		(* CASE AT GLUE GOES FALSE WHEN AXIS IS MOVING AND MODULO GOES OUT OF RANGE *)
		IF (os_case_at_glue_latch OR ls_case_at_glue_latch)
			AND axis_is_moving(csp_case_transport_os_trailing.axis) 
			AND axis_get_actual_modulo_position(csp_case_transport_os_trailing.axis) > glue_trailing_upper_off //unlatch case at glue when past trailing glue flap window
			OR NOT axis_is_cam_engaged(csp_case_transport_os_trailing.axis)
			OR (csp.o_machine_is_stopped
			AND NOT axis_is_moving(csp_case_virtualMaster.axis))//unlatch on stop since glue will dry before closing
		THEN
			os_case_at_glue_latch := FALSE;
			ls_case_at_glue_latch := FALSE;
		END_IF
		
		IF toggle_shift_reg 
			AND	
			shift_register_step_has_status_item(
			step_id := case_at_glue_sr,
			status_bits_to_be_true := ITEM_HAS_LOAD,
			status_bits_to_be_false := 0,
			CONVERSION_this :=csp_case_main_statistics.sr)
		THEN 
			glue_shift_active :=TRUE;
		ELSE
			glue_shift_active :=FALSE;
		END_IF				
	
		
	(* RUN CONDITIONS *)
		IF run_conditions
			AND axis_is_moving(csp_case_transport_os_trailing.axis)
		THEN
			(* CHECKS PHASE WINDOWS TO DETERMINE IF GLUE GUN SHOULD BE ON *)
			
			(* OS UPPER DOTS *)
			IF os_case_at_glue_latch
				AND (
						(dot_1_enable AND phase_window_position_is_in_window(axis_get_actual_modulo_position(csp_case_transport_os_trailing.axis), os_leading_upper_dot_1_phwin)) (* LEADING UPPER DOT 1 *)
						OR (dot_2_enable AND phase_window_position_is_in_window(axis_get_actual_modulo_position(csp_case_transport_os_trailing.axis), os_leading_upper_dot_2_phwin)) (* LEADING UPPER DOT 2 *)
						OR (dot_3_enable AND phase_window_position_is_in_window(axis_get_actual_modulo_position(csp_case_transport_os_trailing.axis), os_leading_upper_dot_3_phwin)) (* LEADING UPPER DOT 3 *)
						OR (dot_4_enable AND phase_window_position_is_in_window(axis_get_actual_modulo_position(csp_case_transport_os_trailing.axis), os_leading_upper_dot_4_phwin)) (* LEADING UPPER DOT 4 *)
						OR (dot_5_enable AND phase_window_position_is_in_window(axis_get_actual_modulo_position(csp_case_transport_os_trailing.axis), os_leading_upper_dot_5_phwin)) (* LEADING UPPER DOT 5 *)
						OR (dot_6_enable AND phase_window_position_is_in_window(axis_get_actual_modulo_position(csp_case_transport_os_trailing.axis), os_leading_upper_dot_6_phwin)) (* LEADING UPPER DOT 6 *)
						OR (dot_1_enable AND phase_window_position_is_in_window(axis_get_actual_modulo_position(csp_case_transport_os_trailing.axis), os_trailing_upper_dot_1_phwin)) (* TRAILING UPPER DOT 1 *)
						OR (dot_2_enable AND phase_window_position_is_in_window(axis_get_actual_modulo_position(csp_case_transport_os_trailing.axis), os_trailing_upper_dot_2_phwin)) (* TRAILING UPPER DOT 2 *)
						OR (dot_3_enable AND phase_window_position_is_in_window(axis_get_actual_modulo_position(csp_case_transport_os_trailing.axis), os_trailing_upper_dot_3_phwin)) (* TRAILING UPPER DOT 3 *)
						OR (dot_4_enable AND phase_window_position_is_in_window(axis_get_actual_modulo_position(csp_case_transport_os_trailing.axis), os_trailing_upper_dot_4_phwin)) (* TRAILING UPPER DOT 4 *)
						OR (dot_5_enable AND phase_window_position_is_in_window(axis_get_actual_modulo_position(csp_case_transport_os_trailing.axis), os_trailing_upper_dot_5_phwin)) (* TRAILING UPPER DOT 5 *)
						OR (dot_6_enable AND phase_window_position_is_in_window(axis_get_actual_modulo_position(csp_case_transport_os_trailing.axis), os_trailing_upper_dot_6_phwin)) (* TRAILING UPPER DOT 6 *)
				)
				AND NOT os_upper_bypass_req
			THEN
					(* OS UPPER GUN 1 IF ENABLED *)
					IF os_upper_gun_1_enable
					THEN
						digital_output_set(os_upper_gun_1_do);
					END_IF
					(* OS UPPER GUN 2 IF ENABLED *)
					IF os_upper_gun_2_enable
					THEN
						digital_output_set(os_upper_gun_2_do);
					END_IF
			ELSE
				digital_output_reset(os_upper_gun_1_do);
				digital_output_reset(os_upper_gun_2_do);
			END_IF
			
			(* OS LOWER DOTS *)
			IF os_case_at_glue_latch
				AND (
						(dot_1_enable AND phase_window_position_is_in_window(axis_get_actual_modulo_position(csp_case_transport_os_trailing.axis), os_leading_lower_dot_1_phwin)) (* LEADING lower DOT 1 *)
						OR (dot_2_enable AND phase_window_position_is_in_window(axis_get_actual_modulo_position(csp_case_transport_os_trailing.axis), os_leading_lower_dot_2_phwin)) (* LEADING lower DOT 2 *)
						OR (dot_3_enable AND phase_window_position_is_in_window(axis_get_actual_modulo_position(csp_case_transport_os_trailing.axis), os_leading_lower_dot_3_phwin)) (* LEADING lower DOT 3 *)
						OR (dot_4_enable AND phase_window_position_is_in_window(axis_get_actual_modulo_position(csp_case_transport_os_trailing.axis), os_leading_lower_dot_4_phwin)) (* LEADING lower DOT 4 *)
						OR (dot_5_enable AND phase_window_position_is_in_window(axis_get_actual_modulo_position(csp_case_transport_os_trailing.axis), os_leading_lower_dot_5_phwin)) (* LEADING lower DOT 5 *)
						OR (dot_6_enable AND phase_window_position_is_in_window(axis_get_actual_modulo_position(csp_case_transport_os_trailing.axis), os_leading_lower_dot_6_phwin)) (* LEADING lower DOT 6 *)
						OR (dot_1_enable AND phase_window_position_is_in_window(axis_get_actual_modulo_position(csp_case_transport_os_trailing.axis), os_trailing_lower_dot_1_phwin)) (* TRAILING lower DOT 1 *)
						OR (dot_2_enable AND phase_window_position_is_in_window(axis_get_actual_modulo_position(csp_case_transport_os_trailing.axis), os_trailing_lower_dot_2_phwin)) (* TRAILING lower DOT 2 *)
						OR (dot_3_enable AND phase_window_position_is_in_window(axis_get_actual_modulo_position(csp_case_transport_os_trailing.axis), os_trailing_lower_dot_3_phwin)) (* TRAILING lower DOT 3 *)
						OR (dot_4_enable AND phase_window_position_is_in_window(axis_get_actual_modulo_position(csp_case_transport_os_trailing.axis), os_trailing_lower_dot_4_phwin)) (* TRAILING lower DOT 4 *)
						OR (dot_5_enable AND phase_window_position_is_in_window(axis_get_actual_modulo_position(csp_case_transport_os_trailing.axis), os_trailing_lower_dot_5_phwin)) (* TRAILING lower DOT 5 *)
						OR (dot_6_enable AND phase_window_position_is_in_window(axis_get_actual_modulo_position(csp_case_transport_os_trailing.axis), os_trailing_lower_dot_6_phwin)) (* TRAILING lower DOT 6 *)
				)
				AND NOT os_lower_bypass_req
			THEN
				(* OS LOWER GUN 1 IF ENABLED *)
				IF os_lower_gun_1_enable
				THEN
					digital_output_set(os_lower_gun_1_do);
				END_IF
				(* OS LOWER GUN 2 IF ENABLED *)
				IF os_lower_gun_2_enable
				THEN
					digital_output_set(os_lower_gun_2_do);
				END_IF
			ELSE
				digital_output_reset(os_lower_gun_1_do);
				digital_output_reset(os_lower_gun_2_do);
			END_IF
			
			
			(* LS UPPER DOTS *)
			IF ls_case_at_glue_latch
				AND (
						(dot_1_enable AND phase_window_position_is_in_window(axis_get_actual_modulo_position(csp_case_transport_ls_trailing.axis), ls_leading_upper_dot_1_phwin)) (* LEADING UPPER DOT 1 *)
						OR (dot_2_enable AND phase_window_position_is_in_window(axis_get_actual_modulo_position(csp_case_transport_ls_trailing.axis), ls_leading_upper_dot_2_phwin)) (* LEADING UPPER DOT 2 *)
						OR (dot_3_enable AND phase_window_position_is_in_window(axis_get_actual_modulo_position(csp_case_transport_ls_trailing.axis), ls_leading_upper_dot_3_phwin)) (* LEADING UPPER DOT 3 *)
						OR (dot_4_enable AND phase_window_position_is_in_window(axis_get_actual_modulo_position(csp_case_transport_ls_trailing.axis), ls_leading_upper_dot_4_phwin)) (* LEADING UPPER DOT 4 *)
						OR (dot_5_enable AND phase_window_position_is_in_window(axis_get_actual_modulo_position(csp_case_transport_ls_trailing.axis), ls_leading_upper_dot_5_phwin)) (* LEADING UPPER DOT 5 *)
						OR (dot_6_enable AND phase_window_position_is_in_window(axis_get_actual_modulo_position(csp_case_transport_ls_trailing.axis), ls_leading_upper_dot_6_phwin)) (* LEADING UPPER DOT 6 *)
						OR (dot_1_enable AND phase_window_position_is_in_window(axis_get_actual_modulo_position(csp_case_transport_ls_trailing.axis), ls_trailing_upper_dot_1_phwin)) (* TRAILING UPPER DOT 1 *)
						OR (dot_2_enable AND phase_window_position_is_in_window(axis_get_actual_modulo_position(csp_case_transport_ls_trailing.axis), ls_trailing_upper_dot_2_phwin)) (* TRAILING UPPER DOT 2 *)
						OR (dot_3_enable AND phase_window_position_is_in_window(axis_get_actual_modulo_position(csp_case_transport_ls_trailing.axis), ls_trailing_upper_dot_3_phwin)) (* TRAILING UPPER DOT 3 *)
						OR (dot_4_enable AND phase_window_position_is_in_window(axis_get_actual_modulo_position(csp_case_transport_ls_trailing.axis), ls_trailing_upper_dot_4_phwin)) (* TRAILING UPPER DOT 4 *)
						OR (dot_5_enable AND phase_window_position_is_in_window(axis_get_actual_modulo_position(csp_case_transport_ls_trailing.axis), ls_trailing_upper_dot_5_phwin)) (* TRAILING UPPER DOT 3 *)
						OR (dot_6_enable AND phase_window_position_is_in_window(axis_get_actual_modulo_position(csp_case_transport_ls_trailing.axis), ls_trailing_upper_dot_6_phwin)) (* TRAILING UPPER DOT 4 *)
				)
				AND NOT ls_upper_bypass_req
			THEN
				(* LS UPPER GUN 1 IF ENABLED *)
				IF ls_upper_gun_1_enable
				THEN
					digital_output_set(ls_upper_gun_1_do);
				END_IF
				(* LS UPPER GUN 2 IF ENABLED *)
				IF ls_upper_gun_2_enable
				THEN
					digital_output_set(ls_upper_gun_2_do);
				END_IF
			ELSE
				digital_output_reset(ls_upper_gun_1_do);
				digital_output_reset(ls_upper_gun_2_do);
			END_IF
			
			(* LS LOWER DOTS *)
			IF ls_case_at_glue_latch
				AND (
						(dot_1_enable AND phase_window_position_is_in_window(axis_get_actual_modulo_position(csp_case_transport_ls_trailing.axis), ls_leading_lower_dot_1_phwin)) (* LEADING lower DOT 1 *)
						OR (dot_2_enable AND phase_window_position_is_in_window(axis_get_actual_modulo_position(csp_case_transport_ls_trailing.axis), ls_leading_lower_dot_2_phwin)) (* LEADING lower DOT 2 *)
						OR (dot_3_enable AND phase_window_position_is_in_window(axis_get_actual_modulo_position(csp_case_transport_ls_trailing.axis), ls_leading_lower_dot_3_phwin)) (* LEADING lower DOT 3 *)
						OR (dot_4_enable AND phase_window_position_is_in_window(axis_get_actual_modulo_position(csp_case_transport_ls_trailing.axis), ls_leading_lower_dot_4_phwin)) (* LEADING lower DOT 4 *)
						OR (dot_5_enable AND phase_window_position_is_in_window(axis_get_actual_modulo_position(csp_case_transport_ls_trailing.axis), ls_leading_lower_dot_5_phwin)) (* LEADING lower DOT 5 *)
						OR (dot_6_enable AND phase_window_position_is_in_window(axis_get_actual_modulo_position(csp_case_transport_ls_trailing.axis), ls_leading_lower_dot_6_phwin)) (* LEADING lower DOT 6 *)
						OR (dot_1_enable AND phase_window_position_is_in_window(axis_get_actual_modulo_position(csp_case_transport_ls_trailing.axis), ls_trailing_lower_dot_1_phwin)) (* TRAILING lower DOT 1 *)
						OR (dot_2_enable AND phase_window_position_is_in_window(axis_get_actual_modulo_position(csp_case_transport_ls_trailing.axis), ls_trailing_lower_dot_2_phwin)) (* TRAILING lower DOT 2 *)
						OR (dot_3_enable AND phase_window_position_is_in_window(axis_get_actual_modulo_position(csp_case_transport_ls_trailing.axis), ls_trailing_lower_dot_3_phwin)) (* TRAILING lower DOT 3 *)
						OR (dot_4_enable AND phase_window_position_is_in_window(axis_get_actual_modulo_position(csp_case_transport_ls_trailing.axis), ls_trailing_lower_dot_4_phwin)) (* TRAILING lower DOT 4 *)
						OR (dot_5_enable AND phase_window_position_is_in_window(axis_get_actual_modulo_position(csp_case_transport_ls_trailing.axis), ls_trailing_lower_dot_5_phwin)) (* TRAILING lower DOT 3 *)
						OR (dot_6_enable AND phase_window_position_is_in_window(axis_get_actual_modulo_position(csp_case_transport_ls_trailing.axis), ls_trailing_lower_dot_6_phwin)) (* TRAILING lower DOT 4 *)
				)
				AND NOT ls_lower_bypass_req
			THEN
				(* LS LOWER GUN 1 IF ENABLED *)
				IF ls_lower_gun_1_enable
				THEN
					digital_output_set(ls_lower_gun_1_do);
				END_IF
				(* LS LOWER GUN 2 IF ENABLED *)
				IF ls_lower_gun_2_enable
				THEN
					digital_output_set(ls_lower_gun_2_do);
				END_IF
			ELSE
				digital_output_reset(ls_lower_gun_1_do);
				digital_output_reset(ls_lower_gun_2_do);
			END_IF
			
			
		ELSE (* LOST RUN CONDITIONS OR GLUE LATCH OR AXIS IS NOT MOVING *)
			(* OS GUNS RESET *)
			digital_output_reset(os_upper_gun_1_do);
			digital_output_reset(os_upper_gun_2_do);
			digital_output_reset(os_lower_gun_1_do);
			digital_output_reset(os_lower_gun_2_do);
			
			(* LS GUNS RESET *)
			digital_output_reset(ls_upper_gun_1_do);
			digital_output_reset(ls_upper_gun_2_do);
			digital_output_reset(ls_lower_gun_1_do);
			digital_output_reset(ls_lower_gun_2_do);
			
			fsm_next_status_NEW := CSP_CASE_GLUE_STATUS_INIT;
		END_IF
				
END_CASE


IF NOT debug_state_machine
	OR
	debug_state_machine_one_step
THEN
	fsm_status_NEW := fsm_next_status_NEW; // TEMP RMH 9.16.2020
	debug_state_machine_one_step := FALSE;
END_IF
END_ACTION

ACTION _set_runtime_properties:
;
END_ACTION

ACTION _write_output:
;
END_ACTION

END_PROGRAM

(* stored: Version 1.1.0.1, ProductVersion 3.1.4024.3
   POU csp_case_glue: Id {7ff7d909-2ce0-4017-86ea-971a1af0a237}, SpecialFunc None
   Action _dot_calculations: Id {278aedba-62c6-063a-096c-418a791e8047}
   Action _handle_messages: Id {3c73a32c-a580-402d-b7b0-44aa52fc39e0}
   Action _handle_process_test: Id {97aebf10-fe30-42a0-aa34-b492b58981d6}
   Action _mode_manager: Id {b4cd57a2-d5f5-43e3-95a4-77dc82d87837}
   Action _object_manager: Id {8a9721d6-db9b-4569-b5ad-18f757257e56}
   Action _read_process_image: Id {813a2253-55f0-454c-a9c3-89d37609ff0a}
   Action _read_var_input: Id {8c837774-6dec-47e8-ac8d-6953eb86a464}
   Action _run_cycle_NEW: Id {41d4716f-73fa-08a5-2b74-e03e1ee2551b}
   Action _set_runtime_properties: Id {b0eca561-6217-4e5d-9c21-f7c76b2529e9}
   Action _write_output: Id {57e3dfe5-204e-4b6a-806b-adebd473ebc7} *)
